FUNCTION MEAN : REAL
VAR_INPUT
    arr : ARRAY[1..10] OF REAL;
END_VAR

VAR
    i : INT;
    sum : REAL := 0.0;
END_VAR

FOR i := 1 TO 10 DO
    sum := sum + arr[i];
END_FOR

MEAN := sum / 10.0;

END_FUNCTION

(* stored: Version 1.1.0.1, ProductVersion 3.1.4024.15
   POU MEAN: Id {75f801e6-40ec-4143-92bf-8eb6093cf0dd}, SpecialFunc None *)
